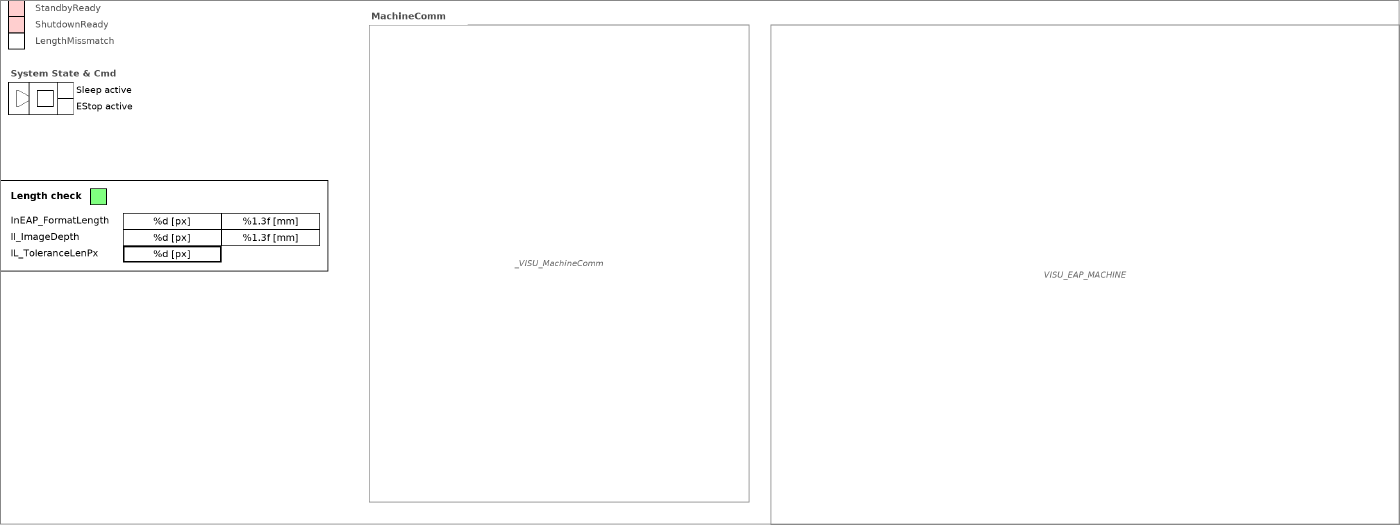
VISUALIZATION VISU_MACHINE  // 1708x641
    Frame (450,30 464x583)
        shows _VISU_MachineComm(mInst := PRG_MACHINE.fbMachineComm)
    Rectangle (450,10 120x20), "MachineComm"
    Rectangle (0,220 400x111)
    Rectangle (270,260 120x20), "%1.3f [mm]", text variable: PRG_MACHINE.InEAP_FormatLength / 1000
    Rectangle (10,260 136x18), "InEAP_FormatLength"
    Rectangle (10,230 96x18), "Length check"
    Rectangle (150,260 120x20), "%d [px]", text variable: PRG_MACHINE.lL_SubstrateLenPx
    Rectangle (270,280 120x20), "%1.3f [mm]", text variable: PRG_PRINT.sAdsPrintUnit[ePr_PU_UNIT_1].sI_JobSettings.lI_ImageDepth / 1000
    Rectangle (10,280 136x18), "lI_ImageDepth"
    Rectangle (150,280 120x20), "%d [px]", text variable: PRG_MACHINE.lL_ImageDepthPx
    RoundedRectangle (110,230 20x20), colour toggle: PRG_MACHINE.bL_MismatchLength
    Rectangle (10,300 136x18), "lL_ToleranceLenPx"
    Rectangle (150,300 120x20), "%d [px]", text variable: PRG_MACHINE.lL_ToleranceLenPx
        OnMouseClick: write the text variable via Default
    Frame (940,30 768x611)
        shows VISU_EAP_MACHINE()
    RoundedRectangle (10,0 20x20)
        toggle PRG_MACHINE.ObEAP_StandbyReady
    Rectangle (40,0 140x20), "StandbyReady"
    RoundedRectangle (10,20 20x20)
        toggle PRG_MACHINE.ObEAP_ShutdownReady
    Rectangle (40,20 140x20), "ShutdownReady"
    RoundedRectangle (10,40 20x20)
        toggle PRG_MACHINE.ObEAP_ShutdownReady
    Rectangle (40,40 140x20), "LengthMissmatch"
    Rectangle (10,80 160x20), "System State & Cmd"
    Group (10,100 20x20), input disabled if: NOT PRG_MACHINE.sADS_Machine[1].sI_Sleep.bO_CommandCanEx
        tap PRG_MACHINE.bL_SleepVisu
        RoundedRectangle (0,0 40x40)
        Polygon (10,10) (12,10) (30,20) (12,30) (10,30)
    Group (35,100 20x20), input disabled if: NOT PRG_MACHINE.sADS_Machine[1].sI_WakeUp.bO_CommandCanEx
        tap PRG_MACHINE.bL_WakeUpVisu
        RoundedRectangle (0,0 40x40)
        Rectangle (10,10 20x20)
    RoundedRectangle (70,100 20x20), colour toggle: PRG_MACHINE.sO_SystemCmd.bSleep
    RoundedRectangle (70,120 20x20), colour toggle: PRG_MACHINE.sO_SystemCmd.bEStop
    RoundedRectangle (90,100 100x20), "Sleep active"
    RoundedRectangle (90,120 100x20), "EStop active"
END_VISUALIZATION

(* stored: Version 1.1.0.1, ProductVersion 3.1.4024.11
   Visu VISU_MACHINE: Id {3edaf7ab-1936-4338-b9d7-1d8cd9d9d5a8} *)
